TYPE U_NCI_R_PARAMETER_Q :
UNION

  stCtrl              : ARRAY[1..MAX_NCI_CH] OF ST_R_Parameter;

  byCtrl    AT %Q*    : ARRAY[1..MAX_NCI_CH] OF
                        ARRAY[1..SIZEOF(ST_R_Parameter)] OF BYTE;
END_UNION
END_TYPE

(* stored: Version 1.1.0.1
   DUT U_NCI_R_PARAMETER_Q: Id {c5a996e1-f8af-4cf7-93d8-dd67b5f6cc75} *)
